FUNCTION AddToStringArray : BOOL
VAR_IN_OUT
	arr : ARRAY[*] OF STRING; //must start from 0 index
END_VAR
VAR_INPUT
	newString : STRING;
END_VAR
VAR_OUTPUT
	numElements : DINT;
	nextIndex : DINT;
END_VAR
VAR
	i : DINT;
END_VAR

FOR i:=LOWER_BOUND(arr, 1) TO UPPER_BOUND(arr, 1) BY 1 DO
	numElements := numElements + 1;
	
	IF arr[i] = '' THEN
		
		arr[i] := newString;
		nextIndex := i + 1;
		
		//ADSLOGSTR(msgCtrlMask := ADSLOG_MSGTYPE_ERROR , msgFmtStr := 'new: %s', strArg := arr[i]);
		
		AddToStringArray := TRUE;
		RETURN;
	END_IF
END_FOR

END_FUNCTION

(* stored: Version 1.1.0.1, ProductVersion 3.1.4024.11
   POU AddToStringArray: Id {62533109-713d-4adc-8713-a6fe80ca70e7}, SpecialFunc None *)
